(* IEC 61131-3 sources: CodesysTest/export/SX_1195.dev/Plc Logic/Application/PRJ Specific/Motion/PLCopen MC, 9 files *)

(* ---- MC_Halt.pou.st ---- *)
(*#-#-#-#-#-#-#-#-#-#---Declaration---#-#-#-#-#-#-#-#-#-#-#-#-#*)

FUNCTION_BLOCK FINAL MC_Halt EXTENDS MC_Base
VAR_INPUT
	deceleration : REAL; 	// Value of the deceleration (decreasing energy of the motor) [u/s²]
END_VAR
VAR_OUTPUT
END_VAR
VAR
END_VAR
(*#-#-#-#-#-#-#-#-#-#---Implementation---#-#-#-#-#-#-#-#-#-#-#-#-#*)

//	Function Block: MC_Halt
//	Description: Commands a controlled motion stop. The axis is moved to the state DiscreteMotion, until the velocity is zero.
//				 When the output Done is set, the state is transferred to Standstill.
//	Created by: Ben Hess
//	Created Date: May 3rd, 2019

//
_executeOSR(CLK := execute);

//
IF _engineState <> eMCEngineState.Idle AND axis.error THEN
	_moveState := eMCMoveState.Error;
	_engineState := eMCEngineState.Idle;
	axis.axisState := eAxisState.Standstill;
	errorID := eMCError.AXIS_ERROR_DURING_COMMAND;
END_IF

//
CASE _engineState OF
	eMCEngineState.Idle:
		IF _executeOSR.Q THEN
			IF NOT axis.error AND axis.operational THEN
				_moveState := eMCMoveState.Busy;
				_engineState := eMCEngineState.Execute;
				errorID := eMCError.NO_ERROR;
			ELSE
				_moveState := eMCMoveState.Error;
				errorID := eMCError.AXIS_NOT_READY;
			END_IF
		END_IF

	eMCEngineState.Execute:
		axis.axisState := eAxisState.Halting;
		axis.halt := TRUE;
		axis.quickStopDeceleration := deceleration;
		_engineState := eMCEngineState.Executing;

	eMCEngineState.Executing:
		axis.halt := FALSE;
		IF axis.actVel = 0 THEN
			_engineState := eMCEngineState.Executed;
		END_IF

	eMCEngineState.Executed:
		axis.axisState := eAxisState.Standstill;
		_moveState := eMCMoveState.Done;
		_engineState := eMCEngineState.Idle;

END_CASE

(* ---- MC_Home.pou.st ---- *)
(*#-#-#-#-#-#-#-#-#-#---Declaration---#-#-#-#-#-#-#-#-#-#-#-#-#*)

FUNCTION_BLOCK FINAL MC_Home EXTENDS MC_Base
VAR_INPUT
END_VAR
VAR_OUTPUT
	homeSuccess : BOOL;
END_VAR
VAR
END_VAR(*#-#-#-#-#-#-#-#-#-#---Implementation---#-#-#-#-#-#-#-#-#-#-#-#-#*)

//	Function Block: MC_Home
//	Description: Commands the axis to perform the «search home» sequence. The details of this sequence are manufacturer specific and can be set by the axis’ parameters.
//				 After completion, the axis state is Standstill if it was Standstill when started.
//	Created by: Ben Hess
//	Created Date: May 3rd, 2019

//
_executeOSR(CLK := execute);

//
IF _engineState <> eMCEngineState.Idle AND axis.error THEN
	_moveState := eMCMoveState.Error;
	_engineState := eMCEngineState.Idle;
	axis.axisState := eAxisState.Standstill;
	errorID := eMCError.AXIS_ERROR_DURING_COMMAND;
END_IF

//
CASE _engineState OF
	eMCEngineState.Idle:
		// Idle State.  If execute rising edge then start halt
		IF NOT execute THEN
			homeSuccess := FALSE;
		END_IF;
		IF _executeOSR.Q THEN
			IF NOT axis.error AND axis.operational THEN
				_moveState := eMCMoveState.Busy;
				_engineState := eMCEngineState.Execute;
				axis.modeOfOperation := eAZDProfileMode.HM;
				errorID := eMCError.NO_ERROR;
			ELSE
				_moveState := eMCMoveState.Error;
				errorID := eMCError.AXIS_NOT_READY;
			END_IF
		END_IF

	eMCEngineState.Execute:
		axis.axisState := eAxisState.Homing;
		axis.startHoming := TRUE;
		_engineState := eMCEngineState.Executing;
		axis.modeOfOperation := eAZDProfileMode.HM;

	eMCEngineState.Executing:
		axis.modeOfOperation := eAZDProfileMode.HM;
		axis.startHoming := FALSE;
		IF axis.isHomed or not execute THEN
			homeSuccess := TRUE;
			_engineState := eMCEngineState.Executed;
		END_IF

	eMCEngineState.Executed:
		_moveState := eMCMoveState.Done;
		_engineState := eMCEngineState.Idle;
		axis.axisState := eAxisState.Standstill;
		axis.modeOfOperation := eAZDProfileMode.PP;

END_CASE

(* ---- MC_MoveAbsolute.pou.st ---- *)
(*#-#-#-#-#-#-#-#-#-#---Declaration---#-#-#-#-#-#-#-#-#-#-#-#-#*)

FUNCTION_BLOCK MC_MoveAbsolute EXTENDS MC_Base
VAR_INPUT
	position : REAL;		// Commanded position for the motion (may be negative) (in technical units [u])
	velocity : REAL;		// Value of the maximum velocity (always positive) (not necessarily reached) [u/s]
	acceleration : REAL;	// Value of the acceleration (always positive) (increasing energy of the motor) [u/s²]
	deceleration : REAL;	// Value of the deceleration (always positive) (decreasing energy of the motor) [u/s²]
	currentLimit : REAL;	// Current limit in %
END_VAR
VAR_OUTPUT
END_VAR
VAR
END_VAR
(*#-#-#-#-#-#-#-#-#-#---Implementation---#-#-#-#-#-#-#-#-#-#-#-#-#*)

//	Function Block: MC_MoveAbsolute
//	Description: Commands a controlled motion to a specified absolute position.
//				 After completion, the axis state is Standstill.
//	Created by: Ben Hess
//	Created Date: May 3rd, 2019

//
_executeOSR(CLK := execute);

//
IF _engineState <> eMCEngineState.Idle AND axis.error THEN
	_moveState := eMCMoveState.Error;
	_engineState := eMCEngineState.Idle;
	errorID := eMCError.AXIS_ERROR_DURING_COMMAND;
END_IF

//
CASE _engineState OF
	eMCEngineState.Idle:
		IF _executeOSR.Q THEN
			IF NOT axis.error AND axis.operational THEN
				_moveState := eMCMoveState.Busy;
				_engineState := eMCEngineState.Execute;
				errorID := eMCError.NO_ERROR;
			ELSE
				_moveState := eMCMoveState.Error;
				errorID := eMCError.AXIS_NOT_READY;
			END_IF
		END_IF

	eMCEngineState.Execute:
		axis.axisState := eAxisState.DiscreteMotion;
		axis.targetPosDist := Position;
		axis.profileVelocity := Velocity;
		axis.profileAcceleration := Acceleration;
		axis.profileDeceleration := Deceleration;
		axis.profileCurrentLimit := currentLimit;
		axis.modeOfOperation := eAZDProfileMode.PP;
		axis.moveAbs := TRUE;
		axis.push := FALSE;
		_engineState := eMCEngineState.Executing;

	eMCEngineState.Executing:
		// Wait for target reached.  Once stopped go back to idle
		axis.moveAbs := FALSE;
		IF axis.targetReached  THEN
			_engineState := eMCEngineState.Executed;
		ELSIF axis.axisState <> eAxisState.DiscreteMotion OR aborted THEN
			_moveState := eMCMoveState.Aborted;
			_engineState := eMCEngineState.Idle;
		END_IF

	eMCEngineState.Executed:
		_moveState := eMCMoveState.Done;
		_engineState := eMCEngineState.Idle;
		axis.axisState := eAxisState.Standstill;

END_CASE

(* ---- MC_MoveAbsolutePush.pou.st ---- *)
(*#-#-#-#-#-#-#-#-#-#---Declaration---#-#-#-#-#-#-#-#-#-#-#-#-#*)

FUNCTION_BLOCK MC_MoveAbsolutePush EXTENDS MC_Base
VAR_INPUT
	position : REAL;		// Commanded position for the motion (may be negative) (in technical units [u])
	velocity : REAL;		// Value of the maximum velocity (always positive) (not necessarily reached) [u/s]
	acceleration : REAL;	// Value of the acceleration (always positive) (increasing energy of the motor) [u/s²]
	deceleration : REAL;	// Value of the deceleration (always positive) (decreasing energy of the motor) [u/s²]
	currentLimit : REAL;	// Current limit in %
END_VAR
VAR_OUTPUT
END_VAR
VAR
END_VAR
(*#-#-#-#-#-#-#-#-#-#---Implementation---#-#-#-#-#-#-#-#-#-#-#-#-#*)

//	Function Block: MC_MoveAbsolute
//	Description: Commands a controlled motion to a specified absolute position.
//				 After completion, the axis state is Standstill.
//	Created by: Ben Hess
//	Created Date: May 3rd, 2019

//
_executeOSR(CLK := execute);

//
IF _engineState <> eMCEngineState.Idle AND axis.error THEN
	_moveState := eMCMoveState.Error;
	_engineState := eMCEngineState.Idle;
	errorID := eMCError.AXIS_ERROR_DURING_COMMAND;
END_IF

//
CASE _engineState OF
	eMCEngineState.Idle:
		IF _executeOSR.Q THEN
			IF NOT axis.error AND axis.operational THEN
				_moveState := eMCMoveState.Busy;
				_engineState := eMCEngineState.Execute;
				errorID := eMCError.NO_ERROR;
			ELSE
				_moveState := eMCMoveState.Error;
				errorID := eMCError.AXIS_NOT_READY;
			END_IF
		END_IF

	eMCEngineState.Execute:
		axis.axisState := eAxisState.DiscreteMotion;
		axis.targetPosDist := Position;
		axis.profileVelocity := Velocity;
		axis.profileAcceleration := Acceleration;
		axis.profileDeceleration := Deceleration;
		axis.modeOfOperation := eAZDProfileMode.PP;
		axis.profilePushCurrentLimit := currentLimit;
		axis.moveAbsTorque := TRUE;
		axis.push := TRUE;
		_engineState := eMCEngineState.Executing;

	eMCEngineState.Executing:
		// Wait for target reached.  Once stopped go back to idle
		axis.moveAbsTorque := FALSE;
		IF axis.targetReached THEN
			_engineState := eMCEngineState.Executed;
		ELSIF axis.axisState <> eAxisState.DiscreteMotion OR aborted THEN
			_moveState := eMCMoveState.Aborted;
			_engineState := eMCEngineState.Idle;
		END_IF

	eMCEngineState.Executed:
		_moveState := eMCMoveState.Done;
		_engineState := eMCEngineState.Idle;
		axis.axisState := eAxisState.Standstill;

END_CASE

(* ---- MC_MoveRelative.pou.st ---- *)
(*#-#-#-#-#-#-#-#-#-#---Declaration---#-#-#-#-#-#-#-#-#-#-#-#-#*)

FUNCTION_BLOCK MC_MoveRelative EXTENDS MC_Base
VAR_INPUT
	distance : REAL;		// Relative distance for the motion (in technical units [u])
	velocity : REAL;		// Value of the maximum velocity (always positive) (not necessarily reached) [u/s]
	acceleration : REAL;	// Value of the acceleration (always positive) (increasing energy of the motor) [u/s²]
	deceleration : REAL;	// Value of the deceleration (always positive) (decreasing energy of the motor) [u/s²]
	currentLimit : REAL;
	torqueModeOnCompletion : BOOL := FALSE;
END_VAR
VAR_OUTPUT
END_VAR
VAR
END_VAR
(*#-#-#-#-#-#-#-#-#-#---Implementation---#-#-#-#-#-#-#-#-#-#-#-#-#*)

//	Function Block: MC_MoveRelative
//	Description: Commands a controlled motion of a specified distance relative to the position at the time of the execution.
//				 The motion completes with velocity zero.
//				 After completion, the axis state is Standstill.
//	Created by: Ben Hess
//	Created Date: May 6th, 2019

IF _engineState <> eMCEngineState.Idle AND axis.error THEN
	_moveState := eMCMoveState.Error;
	_engineState := eMCEngineState.Idle;
	axis.axisState := eAxisState.ErrorStop;
	errorID := eMCError.AXIS_ERROR_DURING_COMMAND;
END_IF

_executeOSR(CLK := execute);
CASE _engineState OF
	eMCEngineState.Idle:
		// Idle State. If execute rising edge then start absolute move
		IF _executeOSR.Q THEN
			IF NOT axis.error AND axis.operational THEN
				_moveState := eMCMoveState.Busy;
				_engineState := eMCEngineState.Execute;
				errorID := eMCError.NO_ERROR;
			ELSE
				_moveState := eMCMoveState.Error;
				errorID := eMCError.AXIS_NOT_READY;
			END_IF
		END_IF

	eMCEngineState.Execute:
		axis.axisState := eAxisState.DiscreteMotion;
		axis.targetPosDist := distance;
		axis.profileVelocity := velocity;
		axis.profileAcceleration := acceleration;
		axis.profileDeceleration := deceleration;
		axis.profileCurrentLimit := currentLimit;
		axis.modeOfOperation := eAZDProfileMode.PP;
		axis.finalMove := torqueModeOnCompletion;
		axis.moveRel := TRUE;
		_engineState := eMCEngineState.Executing;

	eMCEngineState.Executing:
		// Wait for target reached.  Once stopped go back to idle
		axis.moveRel := FALSE;
		IF axis.targetReached THEN
			_engineState := eMCEngineState.Executed;
		ELSIF axis.axisState <> eAxisState.DiscreteMotion OR Aborted OR NOT execute THEN
			_moveState := eMCMoveState.Aborted;
			_engineState := eMCEngineState.Idle;
		END_IF

	eMCEngineState.Executed:
		_moveState := eMCMoveState.Done;
		_engineState := eMCEngineState.Idle;
		axis.axisState := eAxisState.Standstill;

END_CASE

(* ---- MC_MoveVelocity.pou.st ---- *)
(*#-#-#-#-#-#-#-#-#-#---Declaration---#-#-#-#-#-#-#-#-#-#-#-#-#*)

FUNCTION_BLOCK MC_MoveVelocity EXTENDS MC_Base
VAR_INPUT
	execute : BOOL; 		// Rising edge: The halt is started
	velocity : REAL;		// Value of the maximum velocity (always positive) (not necessarily reached) [u/s]
	acceleration : REAL;	// Value of the acceleration (always positive) (increasing energy of the motor) [u/s²]
	deceleration : REAL;	// Value of the deceleration (always positive) (decreasing energy of the motor) [u/s²]
END_VAR
VAR_OUTPUT
	inVelocity : BOOL;		// Value of the commanded velocity (may be negative) (not necessarily reached) [u/s]
	errorID : eMCError;		// Error number
END_VAR
VAR
	_velocityONS : Standard.F_TRIG;
END_VAR
VAR_IN_OUT
	axis : Axis_REF;		// Reference to the axis
END_VAR
(*#-#-#-#-#-#-#-#-#-#---Implementation---#-#-#-#-#-#-#-#-#-#-#-#-#*)

//	Function Block: MC_MoveVelocity
//	Description: Commands a never ending controlled motion with a specified velocity.
//				 To stop the motion, the motion has to be interrupted by another motion command.
//				 The output InVelocity is reset when the block is aborted by another block.
//	Created by: Ben Hess
//	Created Date: May 6th, 2019

//
_velocityONS(CLK := axis.inVelocity);

//
_executeOSR(CLK := execute);

//
IF _engineState <> eMCEngineState.Idle AND axis.error THEN
	_moveState := eMCMoveState.Error;
	_engineState := eMCEngineState.Idle;
	axis.axisState := eAxisState.ErrorStop;
	errorID := eMCError.AXIS_ERROR_DURING_COMMAND;
END_IF

//
CASE _engineState OF
	eMCEngineState.Idle:
		// Idle State.  If execute rising edge then start absolute move
		IF _executeOSR.Q THEN
			IF NOT axis.Error AND axis.operational THEN
				_moveState := eMCMoveState.Busy;
				_engineState := eMCEngineState.Executing;
				errorID := eMCError.NO_ERROR;
			ELSE
				_moveState := eMCMoveState.Error;
				errorID := eMCError.AXIS_NOT_READY;
			END_IF
		END_IF

	eMCEngineState.Execute:
		//
		inVelocity := TRUE;
		axis.axisState := eAxisState.ContinuousMotion;
		axis.profileVelocity := velocity;
		axis.profileAcceleration := acceleration;
		axis.profileDeceleration := deceleration;
		axis.modeOfOperation := eAZDProfileMode.PV;
		axis.moveVel := TRUE;
		_engineState := eMCEngineState.Executing;

	eMCEngineState.Executing:
		axis.moveVel := FALSE;
		IF _velocityONS.Q THEN
			_engineState := eMCEngineState.Executed;
		END_IF

	eMCEngineState.Executed:
		InVelocity := FALSE;
		_engineState := eMCEngineState.Idle;

END_CASE

(* ---- MC_Power.pou.st ---- *)
(*#-#-#-#-#-#-#-#-#-#---Declaration---#-#-#-#-#-#-#-#-#-#-#-#-#*)

FUNCTION_BLOCK MC_Power
VAR_INPUT
	enable : BOOL; 			// Enables the FUNCTION block
END_VAR
VAR_OUTPUT
	status : BOOL; 				// Axis ready for motion
	busy : BOOL; 				// Function block is executing
	error : BOOL; 				// Signals that an error has occured
	errorID : eMCError; 		// Error number
END_VAR
VAR_IN_OUT
	axis : Axis_REF;		// Reference to the axis
END_VAR
(*#-#-#-#-#-#-#-#-#-#---Implementation---#-#-#-#-#-#-#-#-#-#-#-#-#*)

//
//  MC_Power
//  Application/Motion Control/PLCOpen MC/MC_Power
//
//  Created by Evan Ische on 6/29/2022.
//  Copyright (C) 2022 Sharp Packaging Systems By Pregis. All rights reserved.
//

//
axis.driveEnable := enable;

(* ---- MC_Reset.pou.st ---- *)
(*#-#-#-#-#-#-#-#-#-#---Declaration---#-#-#-#-#-#-#-#-#-#-#-#-#*)

FUNCTION_BLOCK FINAL MC_Reset EXTENDS MC_Base
VAR_INPUT
END_VAR
VAR_OUTPUT
END_VAR
VAR
END_VAR(*#-#-#-#-#-#-#-#-#-#---Implementation---#-#-#-#-#-#-#-#-#-#-#-#-#*)

//	Function Block: MC_Reset
//	Description: Forces the transition from the state ErrorStop to Standstill or PowerOff by resetting all internal axis-related errors.
//				 If the axis is not in state ErrorStop, the function block signals the error R_NO_ERROR_TO_RESET.
//	Created by: Ben Hess
//	Created Date: May 14th, 2019

//
_executeOSR(CLK := execute);

//
IF _engineState <> eMCEngineState.Idle AND axis.error THEN
	//_moveState := eMCMoveState.Error;
	//_engineState := eMCEngineState.Idle;
	errorID := eMCError.AXIS_ERROR_DURING_COMMAND;
END_IF

//
CASE _engineState OF
	eMCEngineState.Idle:
		// Idle State.  If execute rising edge then start halt
		IF _executeOSR.Q THEN
			axis.ackError := TRUE;
			_moveState := eMCMoveState.Busy;
			_engineState := eMCEngineState.Execute;
			errorID := eMCError.NO_ERROR;
		END_IF

	eMCEngineState.Execute:
		_engineState := eMCEngineState.Executing;

	eMCEngineState.Executing:

		IF NOT axis.error OR NOT execute THEN
			axis.ackError := FALSE;
			_engineState := eMCEngineState.Executed;
		END_IF

	eMCEngineState.Executed:
		axis.axisState := eAxisState.Standstill;
		_moveState := eMCMoveState.Done;
		_engineState := eMCEngineState.Idle;
END_CASE

(* ---- MC_Stop.pou.st ---- *)
(*#-#-#-#-#-#-#-#-#-#---Declaration---#-#-#-#-#-#-#-#-#-#-#-#-#*)

FUNCTION_BLOCK FINAL MC_Stop EXTENDS MC_Base
VAR_INPUT
	Deceleration : REAL; 	// Value of the deceleration (decreasing energy of the motor) [u/s²]
END_VAR
VAR_OUTPUT
END_VAR
VAR
END_VAR
(*#-#-#-#-#-#-#-#-#-#---Implementation---#-#-#-#-#-#-#-#-#-#-#-#-#*)

//	Function Block: MC_Stop
//	Description: Commands a controlled motion stop. The axis is moved to the state DiscreteMotion, until the velocity is zero.
//				 When the output Done is set, the state is transferred to Standstill.
//	Created by: Ben Hess
//	Created Date: May 3rd, 2019

//
_executeOSR(CLK := execute);

//
IF _engineState <> eMCEngineState.Idle AND axis.error THEN
	_moveState := eMCMoveState.Error;
	_engineState := eMCEngineState.Idle;
	axis.axisState := eAxisState.Standstill;
	errorID := eMCError.AXIS_ERROR_DURING_COMMAND;
END_IF

//
CASE _engineState OF
	eMCEngineState.Idle:
		IF _executeOSR.Q THEN
			IF NOT axis.error AND axis.operational THEN
				_moveState := eMCMoveState.Busy;
				_engineState := eMCEngineState.Execute;
				errorID := eMCError.NO_ERROR;
			ELSE
				_moveState := eMCMoveState.Error;
				errorID := eMCError.AXIS_NOT_READY;
			END_IF
		END_IF

	eMCEngineState.Execute:
		axis.axisState := eAxisState.Halting;
		axis.quickStopDeceleration := deceleration;
		axis.halt := TRUE;
		_engineState := eMCEngineState.Executing;

	eMCEngineState.Executing:
		axis.halt := FALSE;
		IF axis.actVel = 0 THEN
			_engineState := eMCEngineState.Executed;
		END_IF

	eMCEngineState.Executed:
		axis.axisState := eAxisState.Standstill;
		_moveState := eMCMoveState.Done;
		_engineState := eMCEngineState.Idle;

END_CASE
